// TIA Portal V16 export
// export: Created 2024-05-10T06:46:45.2154447Z, ExportSetting WithDefaults, DisplayName Totally Integrated Automation Portal, DisplayVersion V16, DisplayName TIA Portal Version Control Interface, DisplayVersion V16, DisplayName TIA Portal Openness, DisplayVersion V16, DisplayName STEP 7 Professional, DisplayVersion V16, DisplayName STEP 7 Safety, DisplayVersion V16, DisplayName WinCC Professional, DisplayVersion V16
VAR_GLOBAL   // PLC tag table "102故障数据变量表"
   HMI总急停报警 AT %MW6000 : Int;
   HMI总光栅报警 AT %MW6002 : Int;
   HMI总安全门报警 AT %MW6004 : Int;
   HMI总其它安全报警 AT %MW6006 : Int;
   HMI总气压报警 AT %MW6008 : Int;
   HMI总滚筒故障1 AT %MW6010 : Int;
   HMI总滚筒故障2 AT %MW6012 : Int;
   HMI总滚筒故障3 AT %MW6014 : Int;
   HMI总滚筒超时1 AT %MW6016 : Int;
   HMI总滚筒超时2 AT %MW6018 : Int;
   HMI总滚筒超时3 AT %MW6020 : Int;
   HMI总变频器故障 AT %MW6022 : Int;
   HMI总变频器未运行故障 AT %MW6024 : Int;
   HMI总变频器过载故障 AT %MW6026 : Int;
   HMI总变频器超时故障 AT %MW6028 : Int;
   HMI阀出动作超时1 AT %MW6030 : Int;
   HMI阀出动作超时2 AT %MW6032 : Int;
   HMI阀出动作超时3 AT %MW6034 : Int;
   HMI阀出动作超时4 AT %MW6036 : Int;
   HMI阀出动作超时5 AT %MW6038 : Int;
   HMI阀回动作超时1 AT %MW6040 : Int;
   HMI阀回动作超时2 AT %MW6042 : Int;
   HMI阀回动作超时3 AT %MW6044 : Int;
   HMI阀回动作超时4 AT %MW6046 : Int;
   HMI阀回动作超时5 AT %MW6048 : Int;
   HMI阀传感器全到位故障1 AT %MW6050 : Int;
   HMI阀传感器全到位故障2 AT %MW6052 : Int;
   HMI阀传感器全到位故障3 AT %MW6054 : Int;
   HMI阀传感器全到位故障4 AT %MW6056 : Int;
   HMI阀传感器全到位故障5 AT %MW6058 : Int;
   HMI阀传感器交叉ON故障1 AT %MW6060 : Int;
   HMI阀传感器交叉ON故障2 AT %MW6062 : Int;
   HMI阀传感器交叉ON故障3 AT %MW6064 : Int;
   HMI阀传感器交叉ON故障4 AT %MW6066 : Int;
   HMI阀传感器交叉ON故障5 AT %MW6068 : Int;
   HMI伺服报警 AT %MW6070 : Int;
   HMI伺服故障 AT %MW6072 : Int;
   HMI伺服未准备好 AT %MW6074 : Int;
   HMI伺服未回零故障 AT %MW6076 : Int;
   HMI伺服未运行故障 AT %MW6078 : Int;
   HM伺服正极限故障 AT %MW6080 : Int;
   HMI伺服负极限故障 AT %MW6082 : Int;
   HMI视觉故障 AT %MW6084 : Int;
   HMI机器人故障 AT %MW6086 : Int;
   HMI通信故障 AT %MW6088 : Int;
   HMI模拟量上极限故障 AT %MW6090 : Int;
   HMI模拟量下极限故障 AT %MW6092 : Int;
   HMI其它类故障 AT %MW6094 : Int;
   HMI传感器故障1 AT %MW6096 : Int;
   HMI传感器故障2 AT %MW6098 : Int;
   HMI传感器故障3 AT %MW6100 : Int;
   HMI传感器故障4 AT %MW6102 : Int;
   HMI传感器故障5 AT %MW6104 : Int;
   HMI传感器故障6 AT %MW6106 : Int;
   HMI动作异常1 AT %MW6108 : Int;
   HMI动作异常2 AT %MW6110 : Int;
   HMI动作异常3 AT %MW6112 : Int;
END_VAR
